// TIA Portal V19 export
DATA_BLOCK "TimerSetpInInteger"   // DB80
{ S7_Optimized_Access := 'TRUE' }
VERSION : 0.0
// stored: AutoNumber false, MemoryReserve 0
   VAR RETAIN
      COUNT_DOWN_TIMER_VALUE : Int;   // ACTUAL TIMER VALUE COUNT DOWN
      TIMER_SETP_ACTUAL_TIMER : Int;   // TIMER SETPOINT ACTUAL TIMER
      D_2 : Int;
      D_3 : Int;
      D_4 : Int;
      D_5 : Int;
      D_6 : Int;
      D_7 : Int;
      D_8 : Int;
      D_9 : Int;
      SETPOINT_TIMER_10 : Int;   // SETP.T10
      SETPOINT_TIMER_11 : Int;   // SETP.T11
      SETPOINT_TIMER_12 : Int;   // SETP.T12
      SETPOINT_TIMER_13 : Int;   // SETP.T13
      SETPOINT_TIMER_14 : Int := 1800;   // SETP.T14 STERILE TIME
      SETPOINT_TIMER_15 : Int := 600;   // SETP.T15 COOLING TIME
      SETPOINT_TIMER_16 : Int := 30;   // SETP.T16 BLOW OUT CONDENSATE
      SETPOINT_TIMER_17 : Int := 200;   // SETP.T17 BLOW OUT AFTER STOP
      SETPOINT_TIMER_18 : Int := 3;   // SETP.T18 DELAY OPEN 01.12
      SETPOINT_TIMER_19 : Int;   // SETP.T19
      SETPOINT_TIMER_20 : Int;   // SETP.T20
      SETPOINT_TIMER_21 : Int;   // SETP.T21
      SETPOINT_TIMER_22 : Int;   // SETP.T22
      SETPOINT_TIMER_23 : Int;   // SETP.T23
      SETPOINT_TIMER_24 : Int;   // SETP.T24
      SETPOINT_TIMER_25 : Int;   // SETP.T25
      SETPOINT_TIMER_26 : Int;   // SETP.T26
      SETPOINT_TIMER_27 : Int := 500;   // SETP.T27 PRERINSE
      SETPOINT_TIMER_28 : Int := 150;   // SETP.T28 DOSING LYE
      SETPOINT_TIMER_29 : Int := 1800;   // SETP.T29 CIRCULATION LYE
      SETPOINT_TIMER_30 : Int := 600;   // SETP.T30 INTERMEDIATE RINSE
      SETPOINT_TIMER_31 : Int := 140;   // SETP.T31 DOSING ACID
      SETPOINT_TIMER_32 : Int := 1200;   // SETP.T32 CIRCULATION ACID
      SETPOINT_TIMER_33 : Int := 1200;   // SETP.T33 FINAL RINSE
      SETPOINT_TIMER_34 : Int := 300;   // SETP.T34 BLOW OUT AFTER CIP
      SETPOINT_TIMER_35 : Int := 5;   // SETP.T35 DELAY ALARM FILLING PRESSURE
      SETPOINT_TIMER_36 : Int := 25;   // SETP.T36 DELAY TT 01.76 BARRIER
      SETPOINT_TIMER_37 : Int := 25;   // SETP.T37 DELAY TT 01.78 BARRIER
      SETPOINT_TIMER_38 : Int := 10;   // SETP.T38 PAUSE TIME AGITATOR
      SETPOINT_TIMER_39 : Int := 10;   // SETP.T39 RUN TIME AGITATOR
      SETPOINT_TIMER_40 : Int := 4;   // SETP.T40 DELAY RESET STOP LIGHT
      SETPOINT_TIMER_41 : Int := 10;   // SETP.T41 DELAY ALARM STEAM
      SETPOINT_TIMER_42 : Int := 10;   // SETP.T42 DELAY ALARM AIR
      SETPOINT_TIMER_43 : Int := 10;   // SETP.T43 DELAY ALARM WATER
      SETPOINT_TIMER_44 : Int := 300;   // SETP.T44 DELAY BEFORE PURGING
      SETPOINT_TIMER_45 : Int := 25;   // SETP.T45 PURGING FILLING LINE
      SETPOINT_TIMER_46 : Int := 120;   // SETP.T46 PAUSE 01.13 PRESTE.
      SETPOINT_TIMER_47 : Int := 1;   // SETP.T47 OPEN 01.13 PRESTE.
      SETPOINT_TIMER_48 : Int := 10;   // SETP.T48 OPEN 01.13 CIP
      SETPOINT_TIMER_49 : Int := 10;   // SETP.T49 OPEN 01.18 CIP
      SETPOINT_TIMER_50 : Int := 5;   // SETP.T50 OPEN 01.24 CIP
      SETPOINT_TIMER_51 : Int := 120;   // SETP.T51 PAUSE BEFORE 01.08 OPEN
      SETPOINT_TIMER_52 : Int := 5;   // SETP.T52 FLIP 01.44 AT STOP FILLING
      SETPOINT_TIMER_53 : Int := 15;   // SETP.T53 DETERGENT CONC OK
      SETPOINT_TIMER_54 : Int := 240;   // SETP.T54 LYE DOSING TOO LONG
      SETPOINT_TIMER_55 : Int := 240;   // SETP.T55 ACID DOSING TOO LONG
      SETPOINT_TIMER_56 : Int := 5;   // SETP.T56
      SETPOINT_TIMER_57 : Int;   // SETP.T57
      SETPOINT_TIMER_58 : Int := 120;   // SETP.T58
      SETPOINT_TIMER_59 : Int := 5;   // SETP.T59
      SETPOINT_TIMER_60 : Int := 3;   // SETP.T60
      D_61 : Int := 3;
      D_62 : Int;
      D_63 : Int;
      D_64 : Int;
      D_65 : Int;
      D_66 : Int;
      D_67 : Int;
      D_68 : Int;
      D_69 : Int;
      D_70 : Int;
   END_VAR
BEGIN
END_DATA_BLOCK
